# EPICS substitutions: apps/CaenHVApp/Db/CaenHV_Test.substitutions
file "db/AS503_Chan.template" {
pattern
    {P,      H,  S,   V}
    {hchv,   2,  00,   0}
    {hchv,   2,  00,   1}
    {hchv,   2,  01,   0}
    {hchv,   2,  01,   1}
    {hchv,   2,  02,   0}
    {hchv,   2,  02,   1}
    {hchv,   2,  03,   0}
    {hchv,   2,  03,   1}
}
